KUKA KRL program: chk_w6_r2_ab.src, chk_w6_r2_ab.dat

--- chk_w6_r2_ab.src ---
&ACCESS RV2
&REL 2
&PARAM TEMPLATE = C:\KRC\Roboter\Template\vorgabe
&PARAM EDITMASK = *
DEF CHK_W6_R2_AB( )
;
;check all dock stationsbefore release the tool
;Please, verify the inputs to each robot
;Verificar as entradas para adaptar à cada robô
;Dock 1 - 161 (GRIPPER R3)
;Dock 2 - 169
;Dock 3 - 177 (GRIPPER R1)
;Dock 4 - 185 (GRIPPER R4)
;Dock 5 - 193 (GRIPPER R2)
;Dock 6 - 201

IF ($IN[838]==TRUE) THEN

$TIMER[10] = 0
$TIMER_STOP[10] = FALSE

wait for (($in[161]) and ($in[169])  and ($IN[177]) and ($IN[185]) and (NOT $in[193]) and (NOT $in[201]) and ($in[219]))
ELSE

$TIMER[10] = 0
$TIMER_STOP[10] = FALSE

wait for (($in[161]) and ($in[169])  and ($IN[177]) and ($IN[185]) and ($in[193]) and (NOT $in[201]) and ($in[219]))

$TIMER_STOP[10] = TRUE
$TIMER[10] = 0

ENDIF

$TIMER_STOP[10] = TRUE
$TIMER[10] = 0

END

--- chk_w6_r2_ab.dat ---
&ACCESS RV2
&REL 2
&PARAM TEMPLATE = C:\KRC\Roboter\Template\vorgabe
&PARAM EDITMASK = *
DEFDAT CHK_W6_R2_AB
;FOLD EXTERNAL DECLARATIONS;%{PE}%MKUKATPBASIS,%CEXT,%VCOMMON,%P
;FOLD GRIPPERTECH EXT
  EXT  H50 (INT:IN, INT:IN ,INT:IN ,GRP_TYP:IN)
;ENDFOLD (GRIPPERTECH EXT)
;FOLD SPOTTECH EXT

;ENDFOLD (SPOTTECH EXT)
;FOLD BASISTECH EXT;%{PE}%MKUKATPBASIS,%CEXT,%VEXT,%P
EXT  BAS (BAS_COMMAND  :IN,REAL  :IN )
DECL INT SUCCESS
;ENDFOLD (BASISTECH EXT)
;FOLD USER EXT;%{E}%MKUKATPUSER,%CEXT,%VEXT,%P
;Make your modifications here

;ENDFOLD (USER EXT)
;ENDFOLD (EXTERNAL DECLARATIONS)
ENDDAT
